// TIA Portal V15.1 export
// export: Created 2024-06-21T08:41:11.0151079Z, ExportSetting WithDefaults, DisplayName Totally Integrated Automation Portal, DisplayVersion V15.1 Update 5, DisplayName TIA Portal Openness, DisplayVersion V15.1 Update 5, DisplayName SINAMICS Startdrive Advanced, DisplayVersion V15.1, DisplayName G130, G150, S120, S150, SINAMICS MV, S210, DisplayVersion V15.1, DisplayName G110M, G120, G120C, G120D, G120P, DisplayVersion V15.1, DisplayName STEP 7 Professional, DisplayVersion V15.1 Update 5, DisplayName STEP 7 Safety, DisplayVersion V15.1, DisplayName WinCC Professional, DisplayVersion V15.1 Update 5, DisplayName SIMATIC Visualization Architect, DisplayVersion V15.1
FUNCTION "LGBChain2W1S-FC302PN-Config" : Void   // FC6603, FBD
TITLE = LMoveEPos-Config / LGBChain2W1S-FC302PN-Config
{ S7_Optimized_Access := 'FALSE' }
AUTHOR : VCC
FAMILY : Config
VERSION : 0.0.0.0
// =============================================================================
// Configuration MoveUnitEpos
// =============================================================================
// stored: AutoNumber false, IsIECCheckEnabled false, SetENOAutomatically False, UDAEnableTagReadback false
   VAR_INPUT
      C_TrainActivatedSet : Bool;   // Config
      C_TrfInSetUsed : Bool;   // Config
      C_TrfOutSetUsed : Bool;   // Config
      C_TrainActivatedRes : Bool;   // Config
      C_TrfInResUsed : Bool;   // Config
      C_TrfOutResUsed : Bool;   // Config
      C_InitDirection : Bool;   // Config
      C_SafetySwNc : Bool;   // Config
      C_SafetySwUsed : Bool;   // Config
      C_MotorProtectionNc : Bool;   // Config
      C_MotorProtectionUsed : Bool;   // Config
      C_BrakeProtectionNc : Bool;   // Config
      C_BrakeProtectionUsed : Bool;   // Config
      C_MotionStopUsed : Bool;   // Config
      C_EnableAlarmHW : Bool;   // Enable Alarm hardware (e.g. safetyswitch, motorprotector, detections) / Config
      C_EnableAlarmTransfer : Bool;   // Enable Alarm transfer (e.g. Transfer in , transfer out) / Config
      C_EnableCheckSpeedOK : Bool;   // Config
      C_NotQuickStop : Bool;   // QuickStop function; When FALSE the QuickStop of the G120 is active / Config
      C_ReleaseBrakeUsed : Bool;   // Release brake used / Config
      C_TrfMaxTime : DInt;   // Maximum Time (x1ms) that the function may run (create Overtime) / Config
      C_TrfMaxTimeAfterOvertime : DInt;   // Maximum Time (x1ms) that the function may run (create Overtime) / Config
      C_HWSubInput : HW_SUBMODULE;   // I/O / Config
      C_HWSubOutput : HW_SUBMODULE;   // I/O / Config
   END_VAR
   VAR_IN_OUT
      IO_Config : "RollerConvConfig";   // Output Word / Config
   END_VAR
BEGIN

REGION Network 1: **** 1 - Inputs **** Move Config
   // Move Config
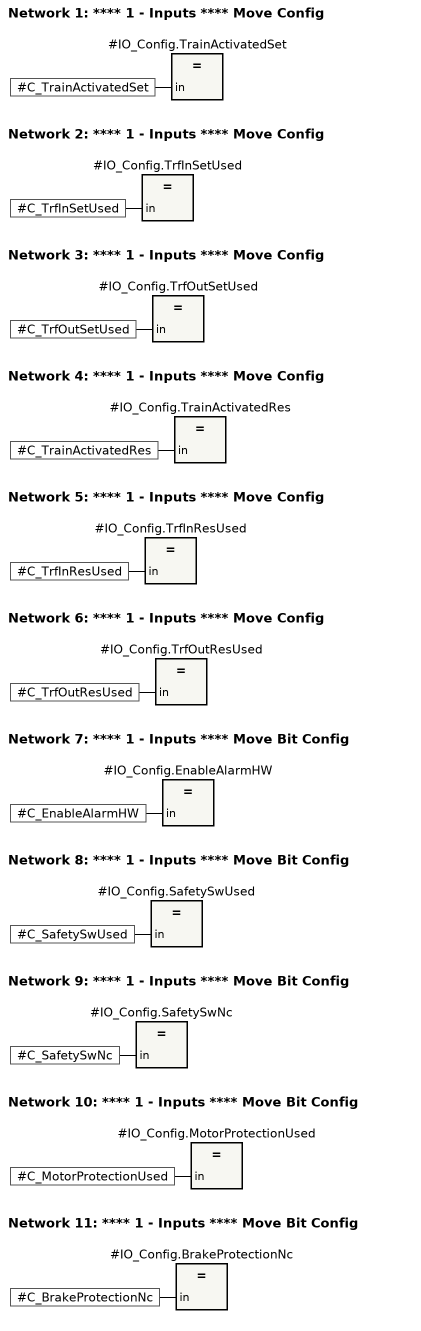
   #IO_Config.TrainActivatedSet := #C_TrainActivatedSet;
END_REGION

REGION Network 2: **** 1 - Inputs **** Move Config
   // Move Config
   #IO_Config.TrfInSetUsed := #C_TrfInSetUsed;
END_REGION

REGION Network 3: **** 1 - Inputs **** Move Config
   // Move Config
   #IO_Config.TrfOutSetUsed := #C_TrfOutSetUsed;
END_REGION

REGION Network 4: **** 1 - Inputs **** Move Config
   // Move Config
   #IO_Config.TrainActivatedRes := #C_TrainActivatedRes;
END_REGION

REGION Network 5: **** 1 - Inputs **** Move Config
   // Move Config
   #IO_Config.TrfInResUsed := #C_TrfInResUsed;
END_REGION

REGION Network 6: **** 1 - Inputs **** Move Config
   // Move Config
   #IO_Config.TrfOutResUsed := #C_TrfOutResUsed;
END_REGION

REGION Network 7: **** 1 - Inputs **** Move Bit Config
   #IO_Config.EnableAlarmHW := #C_EnableAlarmHW;
END_REGION

REGION Network 8: **** 1 - Inputs **** Move Bit Config
   #IO_Config.SafetySwUsed := #C_SafetySwUsed;
END_REGION

REGION Network 9: **** 1 - Inputs **** Move Bit Config
   #IO_Config.SafetySwNc := #C_SafetySwNc;
END_REGION

REGION Network 10: **** 1 - Inputs **** Move Bit Config
   #IO_Config.MotorProtectionUsed := #C_MotorProtectionUsed;
END_REGION

REGION Network 11: **** 1 - Inputs **** Move Bit Config
   #IO_Config.BrakeProtectionNc := #C_BrakeProtectionNc;
END_REGION

REGION Network 12: **** 1 - Inputs **** Move Bit Config
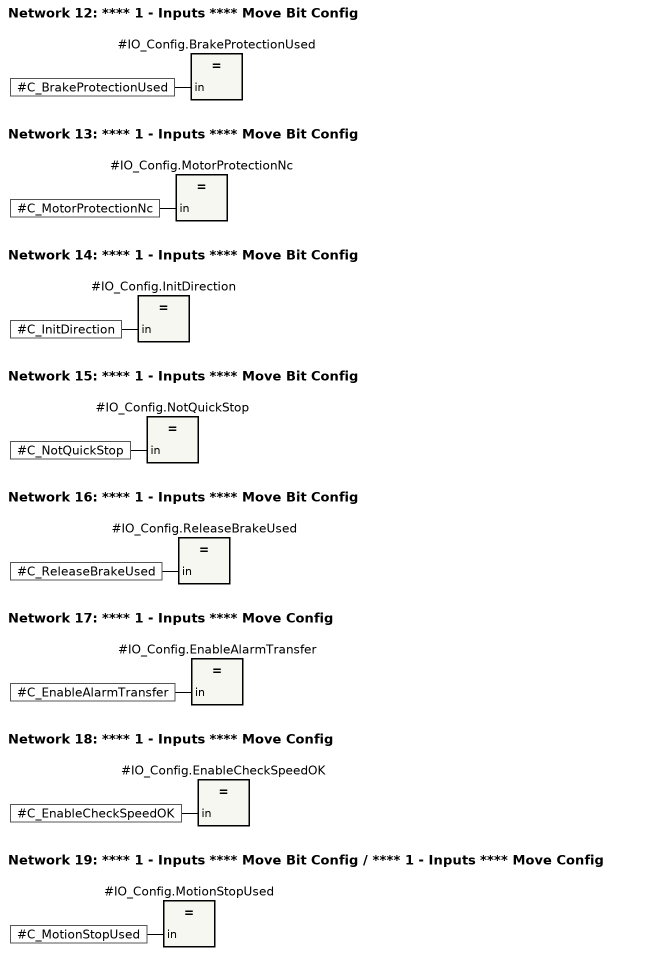
   #IO_Config.BrakeProtectionUsed := #C_BrakeProtectionUsed;
END_REGION

REGION Network 13: **** 1 - Inputs **** Move Bit Config
   #IO_Config.MotorProtectionNc := #C_MotorProtectionNc;
END_REGION

REGION Network 14: **** 1 - Inputs **** Move Bit Config
   #IO_Config.InitDirection := #C_InitDirection;
END_REGION

REGION Network 15: **** 1 - Inputs **** Move Bit Config
   #IO_Config.NotQuickStop := #C_NotQuickStop;
END_REGION

REGION Network 16: **** 1 - Inputs **** Move Bit Config
   #IO_Config.ReleaseBrakeUsed := #C_ReleaseBrakeUsed;
END_REGION

REGION Network 17: **** 1 - Inputs **** Move Config
   // Move Config
   #IO_Config.EnableAlarmTransfer := #C_EnableAlarmTransfer;
END_REGION

REGION Network 18: **** 1 - Inputs **** Move Config
   // Move Config
   #IO_Config.EnableCheckSpeedOK := #C_EnableCheckSpeedOK;
END_REGION

REGION Network 19: **** 1 - Inputs **** Move Bit Config / **** 1 - Inputs **** Move Config
   // Move Bit Config / Move Config
   #IO_Config.MotionStopUsed := #C_MotionStopUsed;
END_REGION

NETWORK
TITLE = **** 1 Inputs **** Move Config UDT
// Move Config
      L     #C_TrfMaxTime;
      T     #IO_Config.TrfMaxTime;
      L     #C_TrfMaxTimeAfterOvertime;
      T     #IO_Config.TrfMaxTimeAfterOvertime;
      L     #C_HWSubInput;
      T     #IO_Config.HWSubInput;
      L     #C_HWSubOutput;
      T     #IO_Config.HWSubOutput;

END_FUNCTION
